TYPE ST_FanucSourceDescriptor :
STRUCT
	MainType : BYTE;
	SubType : BYTE;
	CNCNo : BYTE;
	PathNo : BYTE;
END_STRUCT
END_TYPE

(* stored: Version 1.1.0.1, ProductVersion 3.1.4024.12
   DUT ST_FanucSourceDescriptor: Id {1ba0763a-033e-0910-1996-0df4ec77a2c5} *)
